FUNCTION_BLOCK Test_TStreamAdd_Read_BOOL EXTENDS T_UnitTestBase
VAR
    Stream  : T_Stream(StreamLength := 2);
    ArgType : E_ArgTypeId := E_ArgTypeId.Type_BOOL;
END_VAR

Stream.Init(2);

// add a bool...
Stream.SetNextArgTypeId(ArgType);
Stream.Add_BOOL(TRUE);

Stream.Seek(0);

// check next arg type is correct...
Assertion.AssertEquals_INT(Expected     := ArgType,
                           Actual       := Stream.GetNextArgTypeId(),
                           VariableName := 'Stream.GetNextArgTypeId()');

// check next value...	
Assertion.AssertEquals_BOOL(Expected     := TRUE,
                            Actual       := Stream.Read_BOOL(),
                            VariableName := 'Stream.Read_BOOL()');

// check we are at the end of the stream..							
Assertion.AssertEquals_UDINT(Expected     := Stream.StreamLength,
                             Actual       := Stream.Position,
                             VariableName := 'Stream.Position');

TestFinished();

END_FUNCTION_BLOCK

(* stored: Version 1.1.0.1, ProductVersion 3.1.4024.6
   POU Test_TStreamAdd_Read_BOOL: Id {59f7eb3e-5126-4343-b43d-83136faeeb3b}, SpecialFunc None *)
